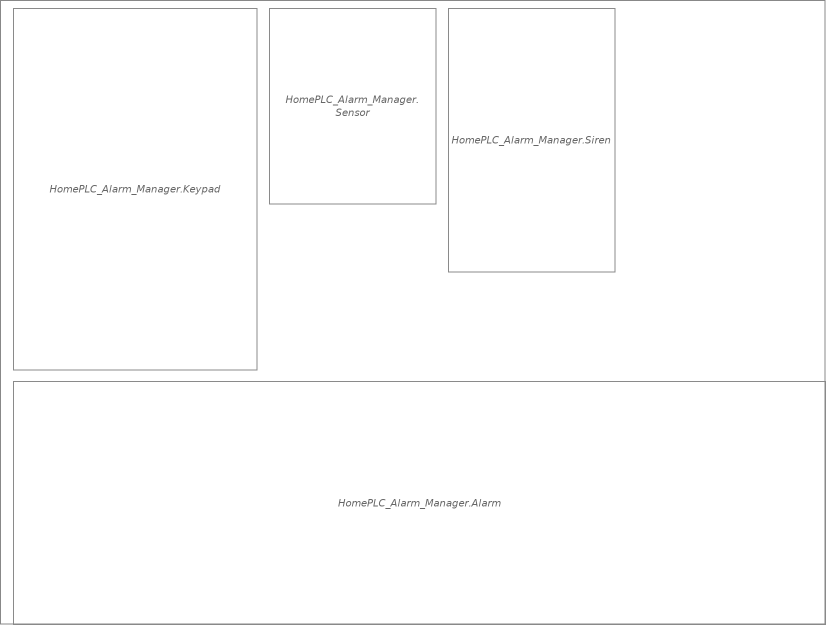
VISUALIZATION Alarm  // 826x625
    Frame (13,8 244x362)
        shows HomePLC_Alarm_Manager.Keypad(stKeypadVirtual := IO.FirstFloor.Entrance.fbAlarmPanel.stVirtual, stKeypad := IO.FirstFloor.Entrance.fbAlarmPanel.stHMI)
    Frame (13,381 813x244)
        shows HomePLC_Alarm_Manager.Alarm(stAlarm := MAIN.fbHome.fbAlarmManager.stHMI)
    Frame (269,8 167x196)
        shows HomePLC_Alarm_Manager.Sensor(stSensor := IO.FirstFloor.Entrance.fbAlarmSensor.stHMI)
    Frame (448,8 167x264)
        shows HomePLC_Alarm_Manager.Siren(stSiren := IO.FirstFloor.Entrance.fbAlarmSiren.stHMI)
END_VISUALIZATION

(* stored: Version 1.1.0.1, ProductVersion 3.1.4024.12
   Visu Alarm: Id {8ec7badd-feaa-4e63-90f1-46cc11bc9ea9} *)
